TYPE TYP_BAN_K50_HW_OUT :
STRUCT
	Red AT %Q* : BOOL;
	Yellow AT %Q* : BOOL;
	Green AT %Q* : BOOL;
END_STRUCT
END_TYPE

(* stored: Version 1.1.0.1, ProductVersion 3.1.4024.12
   DUT TYP_BAN_K50_HW_OUT: Id {494a52b3-fc34-4ef6-8870-1186ee131c87} *)
